// TIA Portal V20 export
// export: Created 2025-12-01T14:57:26.8029459Z, ExportSetting None, DisplayName Totally Integrated Automation Portal, DisplayVersion V20 Update 3, DisplayName TIA Portal Openness, DisplayVersion V20 Update 3, DisplayName TIA Portal Version Control Interface, DisplayVersion V20 Update 3, DisplayName STEP 7 Professional, DisplayVersion V20 Update 3, DisplayName STEP 7 Safety, DisplayVersion V20 Update 2, DisplayName WinCC Basic/Comfort/Advanced, DisplayVersion V20 Update 3, DisplayName WinCC Professional, DisplayVersion V20 Update 3, DisplayName WinCC Unified, DisplayVersion V20 Update 3
FUNCTION "FC605_EventosRec_Quimarox" : Void   // FC605, LAD
{ S7_Optimized_Access := 'FALSE' }
// stored: AutoNumber false, SetENOAutomatically false
   VAR_INPUT
      NumJdT : UInt;   // Numero de JdT recibido el Evento
   END_VAR
   VAR_IN_OUT
      P_Eventos : DWord;   // Puntero al DB de Eventos Recibidos
   END_VAR
   VAR_TEMP
      DBEventosRec : Word;   // DB de Eventos Recibidos
      VarTempQuimarox : Struct
         Quimarox : UInt;
         Mesa : UInt;
      END_STRUCT;
      AtributosDeQuimarox : Struct
         DatosVagon : "CBS_Carrier";
         Mesa : UInt;
         Vagon : UInt;
      END_STRUCT;
      Evento : DWord;   // Etiqueta - Evento
      Atributo : DWord;   // Etiqueta - Atributo
      EtiquetaAtributo : DWord;   // Etiqueta - Conversion de Atributo
      NumeroEvento : UInt;   // Numero de Evento
      NumeroAtributo : UInt;   // Numero de Atributo
      Indice : UInt;
      Leido : UInt;
      OffsetInicial : UInt;
      ValorDeAtributo : UDInt;   // Valor del Atributo
      ReturnValor : Int;
      Cero : Byte;
   END_VAR
BEGIN

NETWORK
TITLE = Inicializar
///////////////////////////////////////////////////////////////////////////////////////////
///////////////////////////////////////////////////////////////////////////////////////////
///////////////////////////////////////////////////////////////////////////////////////////
/// Datos del DB de Recepcion de los Eventos
      L     "JDT1_NDB_EventosRec";  // Cogemos el DB de Eventos Recibidos
      T     #DBEventosRec;

/// --- Comprobar que JDT a enviado el Evento

      L     #NumJdT;
      L     2;
      <>I;
      JC    NoRecibido_JdT02;

      L     "JDT2_NDB_EventosRec";  // Cogemos el DB de Eventos Recibidos
      T     #DBEventosRec;

NoRecibido_JdT02:NOP   0;



NETWORK
TITLE = Distribucion de los Eventos (LIsta del DB de Conversion)
/////////////////////////////////////////////////////////////////////////
/////////////////////////////////////////////////////////////////////////
/////////////////////////////////////////////////////////////////////////
// Hay que recoger el Evento, para despues repartir
// Despues '{' va el tipo de eventos (2 Bytes)
      L     #P_Eventos;  // Recogo por donde va empieza el evento
      LAR2;  // del Quimarox

      OPN   DB [#DBEventosRec];
      L     DBD [AR2, P#0.0];  // Recogo el tipo de Evento (4 Caracteres)
      T     #Evento;


/////////////////////////////////////////////////////////////////////////
/////////////////////////////////////////////////////////////////////////
/////////////////////////////////////////////////////////////////////////
// Buscar numero de evento
      L     1;
      T     #NumeroEvento;
BucleDeBusqueda_NumeroDeEvento:NOP   0;

// -- Se ha encontrado el Evento Recibido
      L     "DB870_ConversorEventos".EventosRecibidos[#NumeroEvento];
      L     #Evento;
      ==D;
      JC    Encontrado_NumeroDeEvento;

// -- Final de la lista de Eventos Recibidos - No Encontrado
      L     "DB870_ConversorEventos".EventosRecibidos[#NumeroEvento];
      L     0;
      ==D;
      JC    NoEncontrado_NumeroDeEvento;

// --- Maximo del Array de la Lista de Eventos Recibidos - No Encontrado
      L     #NumeroEvento;
      L     "CTE_MaxArrayConversion";
      >=I;
      JC    NoEncontrado_NumeroDeEvento;

// --- Continuar la Busqueda
      L     #NumeroEvento;
      L     1;
      +I;
      T     #NumeroEvento;
      JU    BucleDeBusqueda_NumeroDeEvento;


/////////////////////////////////////////////////////////////////////////
// No es ninguno de los eventos previstos, se pasa a buscar el siguiente
NoEncontrado_NumeroDeEvento:NOP   0;
      TAR2;  // Devuelve por donde va empieza el evento
      T     #P_Eventos;  // del Quimarox
      JU    Final_ListaEventos;



NETWORK
TITLE = ----
/////////////////////////////////////////////////////////////////////////
/////////////////////////////////////////////////////////////////////////
/////////////////////////////////////////////////////////////////////////
// Distribuir dependiendo del Resultado de la Busqueda del Evento Recibido
// Para recoger los Atributos
Encontrado_NumeroDeEvento:NOP   0;
      L     #NumeroEvento;
      JL    NoExiste_NumeroDeEvento;

      JU    NoExiste_NumeroDeEvento;
      JU    NoExiste_NumeroDeEvento;  // Evento (01) - CREA
      JU    NoExiste_NumeroDeEvento;  // Evento (02) - RUTA
      JU    NoExiste_NumeroDeEvento;  // Evento (03) - DRUT
      JU    NoExiste_NumeroDeEvento;  // Evento (04) - RETI
      JU    NoExiste_NumeroDeEvento;  // Evento (05) - BORR
      JU    NoExiste_NumeroDeEvento;  // Evento (06) - DATA
      JU    NoExiste_NumeroDeEvento;  // Evento (07) - ?UT?
      JU    NoExiste_NumeroDeEvento;  // Evento (08) - MOVE
      JU    NoExiste_NumeroDeEvento;  // Evento (09) - DEMB
      JU    NoExiste_NumeroDeEvento;  // Evento (10) - CSTA
      JU    NoExiste_NumeroDeEvento;  // Evento (11) - DIDO
      JU    NoExiste_NumeroDeEvento;  // Evento (12) - ORDE
      JU    NoExiste_NumeroDeEvento;  // Evento (13) - BOET
      JU    NoExiste_NumeroDeEvento;  // Evento (14) - BOBD
      JU    NoExiste_NumeroDeEvento;  // Evento (15) - RUET
      JU    NoExiste_NumeroDeEvento;  // Evento (16) - RUES
      JU    NoExiste_NumeroDeEvento;  // Evento (17) - INIR
      JU    NoExiste_NumeroDeEvento;  // Evento (18) - ?ST?

      JU    Atributos_EventosDeQuimarox;  // Evento (19) - QCRE
      JU    Atributos_EventosDeQuimarox;  // Evento (20) - QPR?

/////////////////////////////////////////////////////////////////////////
NoExiste_NumeroDeEvento:NOP   0;
      TAR2;  // Devuelve por donde va empieza el evento
      T     #P_Eventos;  // del Router
      JU    Final_ListaEventos;



NETWORK
TITLE = ////////////////////////////////////////////////////////////////////////////////////////////////////////////

NETWORK
TITLE = Analizar la lista de los Atributos del Quimarox
Atributos_EventosDeQuimarox:NOP   0;

/////////////////////////////////////////////////////////////////////////
/////////////////////////////////////////////////////////////////////////
/////////////////////////////////////////////////////////////////////////
// Inicializa variables de los Atributos de Quimarox
      L     0;
      T     #Cero;

      CALL  FILL
      ( BVAL    := #Cero,
        RET_VAL := #ReturnValor,
        BLK     := #AtributosDeQuimarox
      );  // Inicializa Atributos



NETWORK
TITLE = ----
/////////////////////////////////////////////////////////////////////////
/////////////////////////////////////////////////////////////////////////
// Buscando Atributos o Final del Evento
      +AR2  P#4.0;  // Prepara Puntero para ver los atributos

InicioBucleAtributos_EventosDeQuimarox:NOP   0;
      OPN   DB [#DBEventosRec];
      L     DBB [AR2, P#0.0];
      T     #Leido;

// Inicio de atributo - Ir a tratar los atributos
      L     #Leido;
      L     '[';  // '[' - Inicio de Atributo
      ==I;  // Atributo del Evento
      JC    EncontradoAtributos_EventosDeQuimarox;

// Fin del Evento
      L     #Leido;
      L     '}';  // '}' - Fin del Evento
      ==I;  // Se acabo el evento
      JC    FinalAtributos_EventosDeQuimarox;


// Sin Mensaje
      L     #Leido;
      L     0;  // No hay mas Mensaje
      ==I;  // Se acabo el evento
      JC    FinalAtributos_EventosDeQuimarox;

      +AR2  P#1.0;  // Seguir buscado atributo
      JU    InicioBucleAtributos_EventosDeQuimarox;


/////////////////////////////////////////////////////////////////////////
/////////////////////////////////////////////////////////////////////////
// Se acaba el Evento - Ir a guardar datos del Evento
FinalAtributos_EventosDeQuimarox:NOP   0;
      TAR2;
      T     #P_Eventos;  // Guardo Por donde voy en la lista de eventos
      JU    GuardarDatos_EventosRecibidos;



NETWORK
TITLE = Distribucion de los Atributos del Quimarox (LIsta del DB de Conversion)
EncontradoAtributos_EventosDeQuimarox:NOP   0;

/////////////////////////////////////////////////////////////////////////
/////////////////////////////////////////////////////////////////////////
/////////////////////////////////////////////////////////////////////////
/////////////////////////////////////////////////////////////////////////
// Mirar que Atributo del Evento  es ?
      +AR2  P#1.0;
      OPN   DB [#DBEventosRec];
      L     DBD [AR2, P#0.0];  // Atributo - 4 Caracteres
      T     #Atributo;

/////////////////////////////////////////////////////////////////////////
/////////////////////////////////////////////////////////////////////////
/////////////////////////////////////////////////////////////////////////
// Buscar numero de Atributo
      L     1;
      T     #NumeroAtributo;
BucleDeBusqueda_NumeroDeAtributoDeQuimarox:NOP   0;

// -- Se ha encontrado el Atributo Recibido
      L     "DB870_ConversorEventos".AtributosRecibidosDeQuimarox[#NumeroAtributo];
      L     #Atributo;
      ==D;
      JC    Encontrado_NumeroDeAtributoDeQuimarox;

// -- Final de la lista de Atributo Recibidos - No Encontrado
      L     "DB870_ConversorEventos".AtributosRecibidosDeQuimarox[#NumeroAtributo];
      L     0;
      ==D;
      JC    InicioBucleAtributos_EventosDeQuimarox;

// --- Maximo del Array de la Lista de Atributo Recibidos - No Encontrado
      L     #NumeroAtributo;
      L     "CTE_MaxArrayConversion";
      >=I;
      JC    InicioBucleAtributos_EventosDeQuimarox;


// --- Continuar la Busqueda
      L     #NumeroAtributo;
      L     1;
      +I;
      T     #NumeroAtributo;
      JU    BucleDeBusqueda_NumeroDeAtributoDeQuimarox;



NETWORK
TITLE = ----
/////////////////////////////////////////////////////////////////////////
/////////////////////////////////////////////////////////////////////////
/////////////////////////////////////////////////////////////////////////
// Distribuir dependiendo del Resultado de la Busqueda de Atributo Recibido
Encontrado_NumeroDeAtributoDeQuimarox:NOP   0;
      L     #NumeroAtributo;
      JL    NoExiste_NumeroDeAtibutoDeQuimarox;

      JU    NoExiste_NumeroDeAtibutoDeQuimarox;
      JU    AtributoDeQuimarox_MESA;  // Atributo (01) - MESA
      JU    AtributoDeQuimarox_PEIN;  // Atributo (02) - PEIN
      JU    AtributoDeQuimarox_MCKY;  // Atributo (03) - MCKY
      JU    AtributoDeQuimarox_ORIG;  // Atributo (04) - ORIG
      JU    AtributoDeQuimarox_DEST;  // Atributo (05) - DEST
      JU    AtributoDeQuimarox_SSCC;  // Atributo (06) - SSCC


/////////////////////////////////////////////////////////////////////////
NoExiste_NumeroDeAtibutoDeQuimarox:NOP   0;
      JU    InicioBucleAtributos_EventosDeQuimarox;



NETWORK
TITLE = ---- ---- Recoger el Atributo de Quimarox - MESA
/////////////////////////////////////////////////////////////////////////
/////////////////////////////////////////////////////////////////////////
/////////////////////////////////////////////////////////////////////////
AtributoDeQuimarox_MESA:NOP   0;
      +AR2  P#5.0;
      TAR2;
      T     #P_Eventos;
      SRD   3;
      T     #OffsetInicial;

// Obtener el Valor del Atributo
      CALL  "FC892_Obtener_ValorDelAtributo"
      ( DB_String := #DBEventosRec,
        OffsetIni := #OffsetInicial,
        Valor     := #ValorDeAtributo
      );

      L     #ValorDeAtributo;  // Lo guardo
      T     #AtributosDeQuimarox.Mesa;

// Continuo con el Evento
      L     #P_Eventos;
      LAR2;
      JU    InicioBucleAtributos_EventosDeQuimarox;



NETWORK
TITLE = ---- ---- Recoger el Atributo de Quimarox - PEIN
/////////////////////////////////////////////////////////////////////////
/////////////////////////////////////////////////////////////////////////
/////////////////////////////////////////////////////////////////////////
AtributoDeQuimarox_PEIN:NOP   0;
      +AR2  P#5.0;
      TAR2;
      T     #P_Eventos;
      SRD   3;
      T     #OffsetInicial;

// Obtener el Valor del Atributo
      CALL  "FC892_Obtener_ValorDelAtributo"
      ( DB_String := #DBEventosRec,
        OffsetIni := #OffsetInicial,
        Valor     := #ValorDeAtributo
      );

      L     #ValorDeAtributo;  // Lo guardo
      T     #AtributosDeQuimarox.Vagon;

// Continuo con el Evento
      L     #P_Eventos;
      LAR2;
      JU    InicioBucleAtributos_EventosDeQuimarox;



NETWORK
TITLE = ---- ---- Recoger el Atributo de Quimarox - MCKY
/////////////////////////////////////////////////////////////////////////
/////////////////////////////////////////////////////////////////////////
/////////////////////////////////////////////////////////////////////////
AtributoDeQuimarox_MCKY:NOP   0;
      +AR2  P#5.0;
      TAR2;
      T     #P_Eventos;
      SRD   3;
      T     #OffsetInicial;

// Obtener el Valor del Atributo
      CALL  "FC892_Obtener_ValorDelAtributo"
      ( DB_String := #DBEventosRec,
        OffsetIni := #OffsetInicial,
        Valor     := #ValorDeAtributo
      );

      L     #ValorDeAtributo;  // Lo guardo
      T     #AtributosDeQuimarox.DatosVagon.DatosCarga.Mckey;

// Continuo con el Evento
      L     #P_Eventos;
      LAR2;
      JU    InicioBucleAtributos_EventosDeQuimarox;



NETWORK
TITLE = ---- ---- Recoger el Atributo de Quimarox - ORIG
/////////////////////////////////////////////////////////////////////////
/////////////////////////////////////////////////////////////////////////
/////////////////////////////////////////////////////////////////////////
AtributoDeQuimarox_ORIG:NOP   0;
      +AR2  P#5.0;
      TAR2;
      T     #P_Eventos;
      SRD   3;
      T     #OffsetInicial;

// Obtener el Valor del Atributo
      CALL  "FC892_Obtener_ValorDelAtributo"
      ( DB_String := #DBEventosRec,
        OffsetIni := #OffsetInicial,
        Valor     := #ValorDeAtributo
      );

      L     #ValorDeAtributo;  // Lo guardo
      T     #AtributosDeQuimarox.DatosVagon.DatosCarga.MesaOrigen;

// Continuo con el Evento
      L     #P_Eventos;
      LAR2;
      JU    InicioBucleAtributos_EventosDeQuimarox;



NETWORK
TITLE = ---- ---- Recoger el Atributo de Quimarox - DEST
/////////////////////////////////////////////////////////////////////////
/////////////////////////////////////////////////////////////////////////
/////////////////////////////////////////////////////////////////////////
AtributoDeQuimarox_DEST:NOP   0;
      +AR2  P#5.0;
      TAR2;
      T     #P_Eventos;
      SRD   3;
      T     #OffsetInicial;

// Obtener el Valor del Atributo
      CALL  "FC892_Obtener_ValorDelAtributo"
      ( DB_String := #DBEventosRec,
        OffsetIni := #OffsetInicial,
        Valor     := #ValorDeAtributo
      );

      L     #ValorDeAtributo;  // Lo guardo
      T     #AtributosDeQuimarox.DatosVagon.DatosCarga.MesaDestino;
      T     #AtributosDeQuimarox.DatosVagon.Destino_principal;

// Continuo con el Evento
      L     #P_Eventos;
      LAR2;
      JU    InicioBucleAtributos_EventosDeQuimarox;



NETWORK
TITLE = ---- ---- Recoger el Atributo deQuimarox - SSCC
/////////////////////////////////////////////////////////////////////////
/////////////////////////////////////////////////////////////////////////
/////////////////////////////////////////////////////////////////////////
AtributoDeQuimarox_SSCC:NOP   0;
      +AR2  P#5.0;
      TAR2;
      T     #P_Eventos;
      SRD   3;
      T     #OffsetInicial;

// Obtener el Valor del Atributo
      CALL  "FC892_Obtener_ValorDelAtributo"
      ( DB_String := #DBEventosRec,
        OffsetIni := #OffsetInicial,
        Valor     := #ValorDeAtributo
      );

      L     #ValorDeAtributo;  // Lo guardo
      T     #AtributosDeQuimarox.DatosVagon.DatosCarga.EtiquetaRouter;

// Continuo con el Evento
      L     #P_Eventos;
      LAR2;
      JU    InicioBucleAtributos_EventosDeQuimarox;



NETWORK
TITLE = ////////////////////////////////////////////////////////////////////////////////////////////////////////////

NETWORK
TITLE = Distribucion para Guardar Datos del Evento Recibido (LIsta del DB de Conversion) ///////
/////////////////////////////////////////////////////////////////////////
/////////////////////////////////////////////////////////////////////////
/////////////////////////////////////////////////////////////////////////
GuardarDatos_EventosRecibidos:NOP   0;
      TAR2;
      T     #P_Eventos;  // Guardo Por donde voy en la lista de eventos

      L     #NumeroEvento;
      JL    NoExiste_GuardarDatos_Eventos;

      JU    NoExiste_GuardarDatos_Eventos;
      JU    NoExiste_GuardarDatos_Eventos;  // Evento (01) - CREA
      JU    NoExiste_GuardarDatos_Eventos;  // Evento (02) - RUTA
      JU    NoExiste_GuardarDatos_Eventos;  // Evento (03) - DRUT
      JU    NoExiste_GuardarDatos_Eventos;  // Evento (04) - RETI
      JU    NoExiste_GuardarDatos_Eventos;  // Evento (05) - BORR
      JU    NoExiste_GuardarDatos_Eventos;  // Evento (06) - DATA
      JU    NoExiste_GuardarDatos_Eventos;  // Evento (07) - ?UT?
      JU    NoExiste_GuardarDatos_Eventos;  // Evento (08) - MOVE
      JU    NoExiste_GuardarDatos_Eventos;  // Evento (09) - DEMB
      JU    NoExiste_GuardarDatos_Eventos;  // Evento (10) - CSTA
      JU    NoExiste_GuardarDatos_Eventos;  // Evento (11) - DIDO
      JU    NoExiste_GuardarDatos_Eventos;  // Evento (12) - ORDE
      JU    NoExiste_GuardarDatos_Eventos;  // Evento (13) - BOET
      JU    NoExiste_GuardarDatos_Eventos;  // Evento (14) - BOBD
      JU    NoExiste_GuardarDatos_Eventos;  // Evento (15) - RUET
      JU    NoExiste_GuardarDatos_Eventos;  // Evento (16) - RUES
      JU    NoExiste_GuardarDatos_Eventos;  // Evento (17) - INIR
      JU    NoExiste_GuardarDatos_Eventos;  // Evento (18) - ?ST?

      JU    GuardarDatos_EventoRecibido_QCRE;  // Evento (19) - QCRE
      JU    GuardarDatos_EventoRecibido_Refresco_Quimarox;  // Evento (20) - QPR?


/////////////////////////////////////////////////////////////////////////
NoExiste_GuardarDatos_Eventos:NOP   0;
      JU    Final_ListaEventos;



NETWORK
TITLE = ////////////////////////////////////////////////////////////////////////////////////////////////////////////

NETWORK
TITLE = Evento QCRE - Crea una Carga en el Vagon del Quimarox
GuardarDatos_EventoRecibido_QCRE:NOP   0;

/////////////////////////////////////////////////////////////////////////
/////////////////////////////////////////////////////////////////////////
/////////////////////////////////////////////////////////////////////////
// --- Guardar Datos del Evento Recibido


/////////////////////////////////////////////////////////////////////////
/////////////////////////////////////////////////////////////////////////
/////////////////////////////////////////////////////////////////////////
/// --- Buscar Numero de Quimarox
      L     1;
      T     #VarTempQuimarox.Quimarox;

      L     #AtributosDeQuimarox.Mesa;
      L     "CTE_OffsetMesa";
      -I;
      T     #VarTempQuimarox.Mesa;

BuscarNumeroQuimarox_EventoRecibido_QCRE:NOP   0;
      L     #VarTempQuimarox.Mesa;  // Mesa Asociada = Mesa Recibida
      L     "DB600_ConfigQuimarox".Quimarox[#VarTempQuimarox.Quimarox].datos_config.Numero_MesaAsociada;
      ==I;
      JC    GuardarDatosVagonQuimarox_EventoRecibido_QCRE;

      L     #VarTempQuimarox.Quimarox;  // Siguiente Quimarox
      L     1;
      +I;
      T     #VarTempQuimarox.Quimarox;

      L     #VarTempQuimarox.Quimarox;  // Existen mas Quimarox
      L     "CTE_MaxNumQuimarox";
      >I;
      JC    Final_EventoRecibido_QCRE;
      JU    BuscarNumeroQuimarox_EventoRecibido_QCRE;



NETWORK
TITLE = ---- Guardar Datos del Vagon del Quimarox
GuardarDatosVagonQuimarox_EventoRecibido_QCRE:NOP   0;

/////////////////////////////////////////////////////////////////////////
/////////////////////////////////////////////////////////////////////////
/////////////////////////////////////////////////////////////////////////
// --- Comprobar si existe Vagon ( 0 > Vagon < Numero de Vagones )
      L     #AtributosDeQuimarox.Vagon;
      L     1;
      <I;
      JC    Final_EventoRecibido_QCRE;
      L     #AtributosDeQuimarox.Vagon;
      L     "DB600_ConfigQuimarox".Quimarox[#VarTempQuimarox.Quimarox].datos_config.Numero_vagones;
      >I;
      JC    Final_EventoRecibido_QCRE;


/////////////////////////////////////////////////////////////////////////
/////////////////////////////////////////////////////////////////////////
/////////////////////////////////////////////////////////////////////////
// --- Guardar Datos del Vagon de quimarox
      SET;
      S     #AtributosDeQuimarox.DatosVagon.Carrier_Cargado;

// --- Inicializar Datos Vagon
      CALL  UBLKMOV
      ( SRCBLK  := #AtributosDeQuimarox.DatosVagon,
        RET_VAL := #ReturnValor,
        DSTBLK  := "DB601_PeinesQuimarox".Quimarox[#VarTempQuimarox.Quimarox].vagon[#AtributosDeQuimarox.Vagon]
      );  // --- Copiar los Datos del Vagon



NETWORK
TITLE = ---- Final
///////////////////////////////////////////////////////////////////////////////
///////////////////////////////////////////////////////////////////////////////
///////////////////////////////////////////////////////////////////////////////
// --- Se acabo el evento
Final_EventoRecibido_QCRE:NOP   0;
      L     #P_Eventos;  // Recupero por donde voy en la lista de eventos
      LAR2;  // Regreso a buscar el siguiente evento
      JU    Final_ListaEventos;



NETWORK
TITLE = ////////////////////////////////////////////////////////////////////////////////////////////////////////////

NETWORK
TITLE = Evento QPR? - Peticion de Datos de los Vagones del Quimarox
// - Inicializa variables de los atributos del Evento
// - Buscar Atributos o Final del Evento
// - Guardar datos del Evento
//   - Si tiene Tipo y Numero
//   - Si solo Tipo
//   - Si son todos
GuardarDatos_EventoRecibido_Refresco_Quimarox:NOP   0;

/////////////////////////////////////////////////////////////////////////
/////////////////////////////////////////////////////////////////////////
/////////////////////////////////////////////////////////////////////////
// --- Guardar Datos del Evento Recibido


/////////////////////////////////////////////////////////////////////////
/////////////////////////////////////////////////////////////////////////
/////////////////////////////////////////////////////////////////////////
/// --- Buscar Numero de Quimarox
      L     1;
      T     #VarTempQuimarox.Quimarox;

      L     #AtributosDeQuimarox.Mesa;
      L     "CTE_OffsetMesa";
      -I;
      T     #VarTempQuimarox.Mesa;

BuscarNumeroQuimarox_EventoRecibido_Refresco_Quimarox:NOP   0;
      L     #VarTempQuimarox.Mesa;  // Mesa Asociada = Mesa Recibida
      L     "DB600_ConfigQuimarox".Quimarox[#VarTempQuimarox.Quimarox].datos_config.Numero_MesaAsociada;
      ==I;
      JC    GuardarDatosVagonQuimarox_EventoRecibido_Refresco_Quimarox;

      L     #VarTempQuimarox.Quimarox;  // Siguiente Quimarox
      L     1;
      +I;
      T     #VarTempQuimarox.Quimarox;

      L     #VarTempQuimarox.Quimarox;  // Existen mas Quimarox
      L     "CTE_MaxNumQuimarox";
      >I;
      JC    Final_EventoRecibido_Refresco_Quimarox;
      JU    BuscarNumeroQuimarox_EventoRecibido_Refresco_Quimarox;



NETWORK
TITLE = ---- Guardar Datos del Vagon del Quimarox
GuardarDatosVagonQuimarox_EventoRecibido_Refresco_Quimarox:NOP   0;

///////////////////////////////////////////////////////////////////////////////
///////////////////////////////////////////////////////////////////////////////
///////////////////////////////////////////////////////////////////////////////
/// --- Guardar los Datos del Vagon
      L     1;
      T     #Indice;

Bucle_GuardarDatosVagonQuimarox_EventoRecibido_Refresco_Quimarox:NOP   0;
      L     "DB601_PeinesQuimarox".Quimarox[#VarTempQuimarox.Quimarox].vagon[#Indice].DatosCarga.Mckey;
      L     0;  // Tiene datos
      ==I;
      JC    SiguienteBucle_GuardarDatosVagon_EventoPeticionDatosVagones;

      L     "CTE_Evento_QPRE";  // Generar Evento
      T     "DB601_PeinesQuimarox".Quimarox[#VarTempQuimarox.Quimarox].vagon[#Indice].EventoAGenerar;

SiguienteBucle_GuardarDatosVagon_EventoPeticionDatosVagones:NOP   0;
      L     #Indice;  // Siguiente Vagon o Hay mas vagones
      L     1;
      +I;
      T     #Indice;

      L     #Indice;
      L     "DB600_ConfigQuimarox".Quimarox[#VarTempQuimarox.Quimarox].datos_config.Numero_vagones;
      >I;
      JC    Final_EventoRecibido_Refresco_Quimarox;
      JU    Bucle_GuardarDatosVagonQuimarox_EventoRecibido_Refresco_Quimarox;



NETWORK
TITLE = ---- Final
///////////////////////////////////////////////////////////////////////////////
///////////////////////////////////////////////////////////////////////////////
///////////////////////////////////////////////////////////////////////////////
// --- Se acabo el evento
Final_EventoRecibido_Refresco_Quimarox:NOP   0;
      L     #P_Eventos;  // Recupero por donde voy en la lista de eventos
      LAR2;  // Regreso a buscar el siguiente evento
      JU    Final_ListaEventos;



NETWORK
TITLE = ////////////////////////////////////////////////////////////////////////////////////////////////////////////

NETWORK
TITLE = Final de la Lista de Eventos
///////////////////////////////////////////////////////////////////////////////////////////
///////////////////////////////////////////////////////////////////////////////////////////
///////////////////////////////////////////////////////////////////////////////////////////
/// Final de la Recepcion de la Lista de Eventos
Final_ListaEventos:NOP   0;


END_FUNCTION
